// TIA Portal V20 export
TYPE "LER_TypeFATMode_Sampling"
// stored: Access Published
   STRUCT
      ProcessValue : "LER_TypeFATMode_Sampling_ProcessValue";
      SetValue : "LER_TypeFATMode_Sampling_SetValue";
   END_STRUCT;
END_TYPE
